(* Logix 5000 project; controller CICD_test 1756-L85E rev 36.11; software revision 36.00 *)

TASK MainTask (continuous, watchdog 500 ms) : MainProgram

MODULES
   Local : 1756-L85E (ICP 0, rev 36.11)
END_MODULES

ADD_ON_INSTRUCTION AOI_Comparison   (* revision 1.0, ExecutePrescan *)
VAR_INPUT
   I_Parameter1 : DINT; {required}
   I_Parameter2 : DINT; {required}
END_VAR
VAR_OUTPUT
   O_Param1_grtr_than_Param2 : BOOL; {visible}
END_VAR

ROUTINE Logic   (* ladder *)
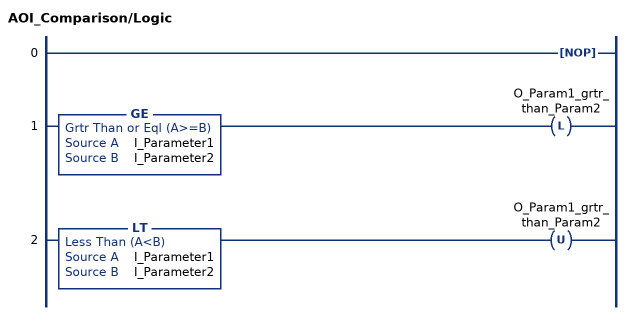
   0: NOP();
   1: GE(I_Parameter1,I_Parameter2)OTL(O_Param1_grtr_than_Param2);
   2: LT(I_Parameter1,I_Parameter2)OTU(O_Param1_grtr_than_Param2);
END_ROUTINE

ROUTINE Prescan   (* ladder *)
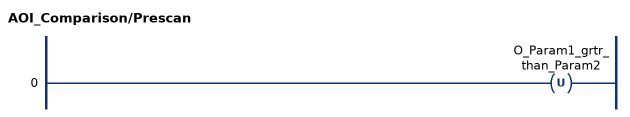
   0: OTU(O_Param1_grtr_than_Param2);
END_ROUTINE
END_ADD_ON_INSTRUCTION

ADD_ON_INSTRUCTION AOI_ModuleReset   (* revision 1.0 JDR *)
// Inhibits Module, Reset Module, Uninhibits Module
// Revision note:
// Developed for Safety I/O module reset with Signature/Lock
// Help:
// Inhibits Module, Reset Module, Uninhibits Module
// msg_Module_Reset can be shared by many modules, but must have Service Type = Device Reset
// The MSG path is set from IO_ModRef inside the AOI.
VAR_IN_OUT
   MSG_Module_Reset : MESSAGE; {required}   // Message Reset Module
   IO_ModRef : MODULE; {required}   // Module Reference
END_VAR
VAR_INPUT
   Cmd_Reset : BOOL; {required}   // Input Command To Run Routine
END_VAR
VAR_OUTPUT
   MSG_Err : BOOL; {access Read Only, visible}   // Message Error
   Mod_Flt : BOOL; {access Read Only, visible}   // Module Faulted
   Mod_Con : BOOL; {access Read Only, visible}   // Module Connecting
   Mod_Run : BOOL; {access Read Only, visible}   // Module Running
END_VAR
VAR
   ModulePath : SINT[82]; {access None}   // Module Path
   ONS : DINT; {access None}   // One Shot Array
   CardInhibit : DINT; {access None}   // Inhibit Value
   CardUnInhibit : DINT; {access None}   // UnInhibit Value
   Module_EntryStatus : DINT; {access None}   // Module Entry Status h1000 = Faulted h3000 = Connecting h4000 = Running h6000 = Inhibitted
   Reset_Run : BOOL; {access None}   // Run Reset Logic
   ModRun_TMR : TIMER := (PRE := 2000); {access None}   // Module Running Timer
   Mod_Inhibitted : BOOL; {access None}   // Module Inhibitted
END_VAR

ROUTINE Logic   (* ladder *)
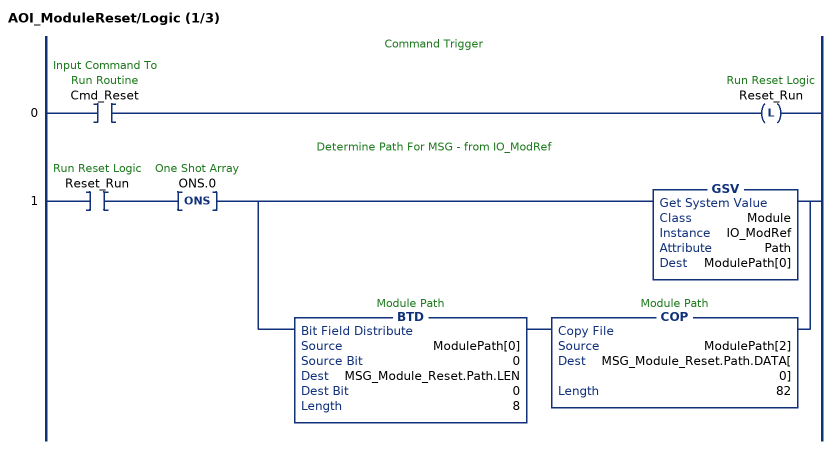
   // Command Trigger
   0: XIC(Cmd_Reset)OTL(Reset_Run);
   // Determine Path For MSG - from IO_ModRef
   1: XIC(Reset_Run)ONS(ONS.0)[GSV(Module,IO_ModRef,Path,ModulePath[0]) ,BTD(ModulePath[0],0,MSG_Module_Reset.Path.LEN,0,8) COP(ModulePath[2],MSG_Module_Reset.Path.DATA[0],82) ];
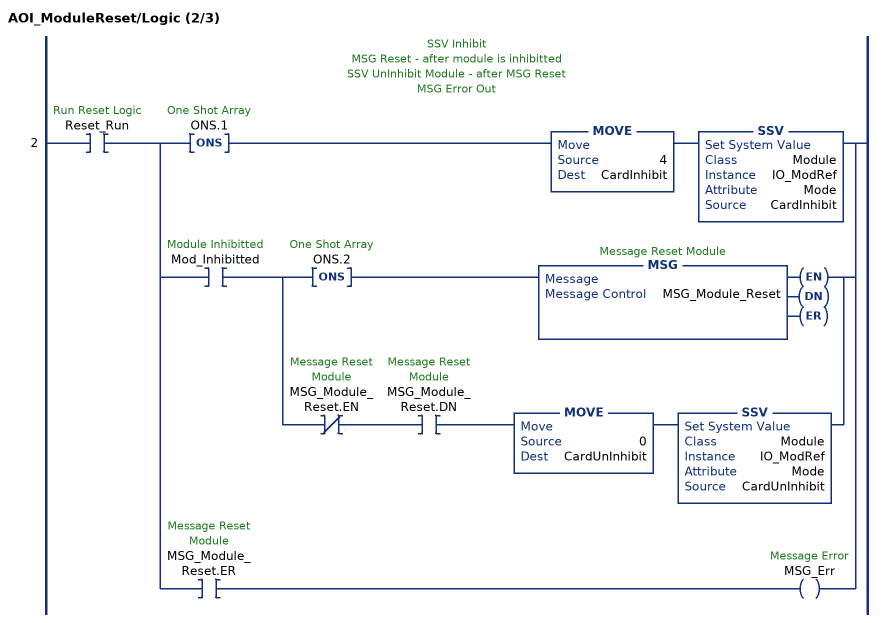
   // SSV Inhibit
   // MSG Reset - after module is inhibitted
   // SSV UnInhibit Module - after MSG Reset
   // MSG Error Out
   2: XIC(Reset_Run)[ONS(ONS.1) MOVE(4,CardInhibit) SSV(Module,IO_ModRef,Mode,CardInhibit) ,XIC(Mod_Inhibitted) [ONS(ONS.2) MSG(MSG_Module_Reset) ,XIO(MSG_Module_Reset.EN) XIC(MSG_Module_Reset.DN) MOVE(0,CardUnInhibit) SSV(Module,IO_ModRef,Mode,CardUnInhibit) ] ,XIC(MSG_Module_Reset.ER) OTE(MSG_Err) ];
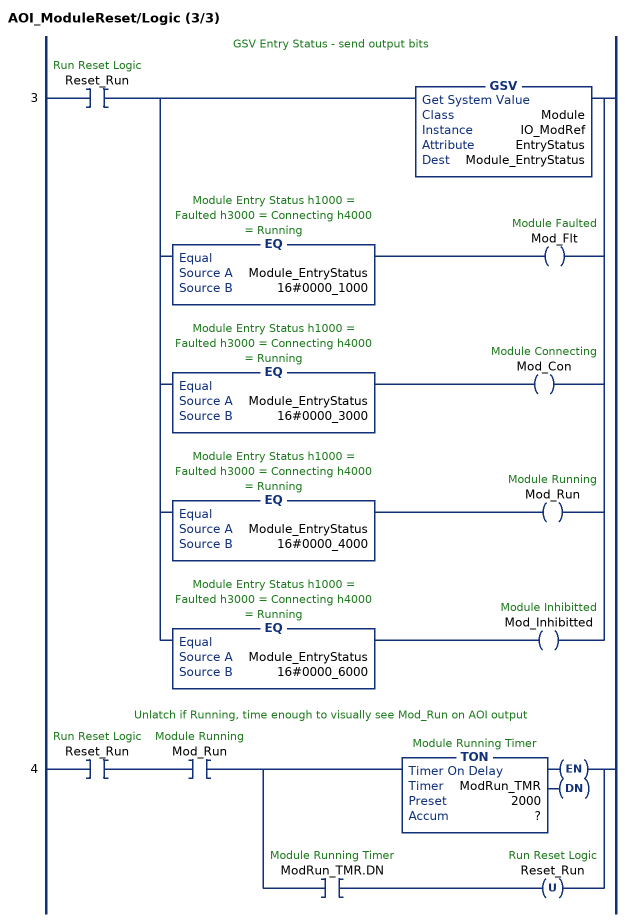
   // GSV Entry Status - send output bits
   3: XIC(Reset_Run)[GSV(Module,IO_ModRef,EntryStatus,Module_EntryStatus) ,EQ(Module_EntryStatus,16#0000_1000) OTE(Mod_Flt) ,EQ(Module_EntryStatus,16#0000_3000) OTE(Mod_Con) ,EQ(Module_EntryStatus,16#0000_4000) OTE(Mod_Run) ,EQ(Module_EntryStatus,16#0000_6000) OTE(Mod_Inhibitted) ];
   // Unlatch if Running, time enough to visually see Mod_Run on AOI output
   4: XIC(Reset_Run)XIC(Mod_Run)[TON(ModRun_TMR,?,?) ,XIC(ModRun_TMR.DN) OTU(Reset_Run) ];
END_ROUTINE
END_ADD_ON_INSTRUCTION

VAR_GLOBAL   (* controller tags *)
   Comparison_AOI : AOI_Comparison := (O_Param1_grtr_than_Param2 := 1);
   O_Comparison_Success : BOOL := 1;
   test_BOOL : BOOL;
   test_DINT_1 : DINT := 2;
   test_DINT_2 : DINT := 20;
   test_DINT_3 : DINT := 30;
   test_STRING : STRING;
END_VAR

PROGRAM MainProgram   (* main routine MainRoutine *)

ROUTINE MainRoutine   (* ladder *)
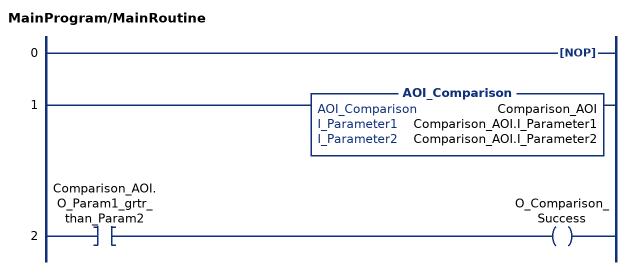
   0: NOP();
   1: AOI_Comparison(Comparison_AOI,Comparison_AOI.I_Parameter1,Comparison_AOI.I_Parameter2);
   2: XIC(Comparison_AOI.O_Param1_grtr_than_Param2)OTE(O_Comparison_Success);
END_ROUTINE
END_PROGRAM
